PROGRAM MAIN
VAR
	MpsLogicUpgrade : MpsLogicUpgrade;
	RtdReadings : RtdReadings;
	//MpsLogicTest : MpsLogicTest;
	
END_VAR

//EPICS test

MpsLogicUpgrade();
RtdReadings();

//MpsLogicTest();

END_PROGRAM

(* stored: Version 1.1.0.1, ProductVersion 3.1.4024.12
   POU MAIN: Id {1f25c106-3603-4b66-a9dc-d624e71d8258}, SpecialFunc None *)
